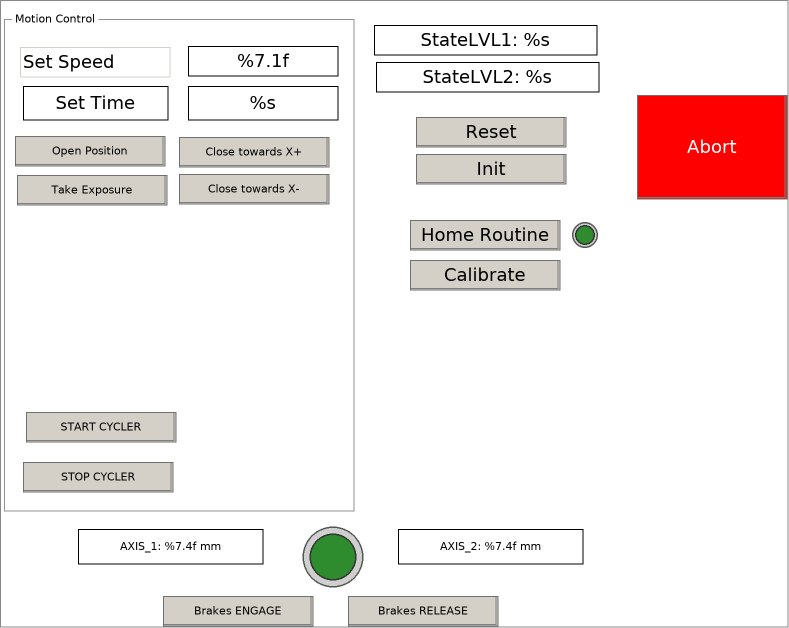
VISUALIZATION ShutterGUI  // 789x628
    GroupBox (4,11 350x500), "Motion Control"
        Rectangle (19,75 145x34), "Set Time", input disabled if: MAIN.shutterFSM.stateLVL2 <> 0;
            OnMouseUp: write GVL.expoTime via Edit, format %7.1f
        Rectangle (184,75 150x34), "%s", text variable: GVL.expoTime
        Button (22,401 150x30), "START CYCLER", input disabled if: MAIN.motionState <> 100;
            OnMouseUp: execute { MAIN.motionState:=3100; }
        Button (19,451 150x30), "STOP CYCLER"
            OnMouseUp: execute { MAIN.stop:=TRUE; }
        Button (13,164 150x30), "Take Exposure", input disabled if: MAIN.shutterFSM.stateLVL2 <> 0;
            OnMouseUp: execute { MAIN.command := commands.takeExposure; }
        Button (11,125 150x30), "Open Position", input disabled if: MAIN.shutterFSM.stateLVL2 <> 0;
            OnMouseUp: execute { MAIN.command := commands.openShutter; }
        Button (175,126 150x30), "Close towards X+", input disabled if: MAIN.shutterFSM.stateLVL2 <> 0;
            OnMouseUp: execute { MAIN.command := commands.closeShutterPX; }
        Button (175,163 150x30), "Close towards X-", input disabled if: MAIN.shutterFSM.stateLVL2 <> 0;
            OnMouseUp: execute { MAIN.command := commands.closeShutterMX; }
    Button (163,596 150x30), "Brakes ENGAGE", input disabled if: MAIN.axis[0].brake=FALSE AND MAIN.axis[1].brake=FALSE;
        OnMouseClick: execute { MAIN.axis[0].brake:=FALSE; MAIN.axis[1].brake:=FALSE; }
    Button (348,596 150x30), "Brakes RELEASE", input disabled if: MAIN.axis[0].brake=TRUE AND MAIN.axis[1].brake=TRUE;
        OnMouseClick: execute { MAIN.axis[0].brake:=TRUE; MAIN.axis[1].brake:=TRUE; }
    Lamp1 (298,522 70x70), variable: MAIN.axis[0].brake and MAIN.axis[1].brake;, style: Lamp-Lamp1-Green
    Rectangle (78,529 185x35), "AXIS_1: %7.4f mm", text variable: MAIN.axis[0].axisRef.NcToPlc.ActPos
    Rectangle (398,529 185x35), "AXIS_2: %7.4f mm", text variable: MAIN.axis[1].axisRef.NcToPlc.ActPos
    Button (416,117 150x30), "Reset"
        OnMouseUp: execute { MAIN.command := commands.clearAllFaults; }
    Button (637,95 150x104), "Abort"
        OnMouseUp: execute { MAIN.command := commands.stopAllMotion; }
    Rectangle (374,25 223x30), "StateLVL1: %s", text variable: MAIN.shutterFSM.stateLVL1;
    Button (410,220 150x30), "Home Routine", input disabled if: MAIN.motionState <> 100;
        OnMouseUp: execute { MAIN.motionState := 400; }
    Textfield (20,47 150x30), "Set Speed", input disabled if: MAIN.shutterFSM.stateLVL2 <> 0;
        OnMouseUp: write MAIN.speed via Default, min 0, max 2000, format %7.1f
    Rectangle (188,46 150x30), "%7.1f", text variable: MAIN.speed
    Lamp1 (570,220 30x30), variable: MAIN.axis[0].axisRef.Status.Homed and MAIN.axis[1].axisRef.Status.Homed;, style: Lamp-Lamp1-Green
    Button (410,260 150x30), "Calibrate", input disabled if: MAIN.motionState <> 100;
        OnMouseUp: execute { MAIN.motionState:=8000; }
    Rectangle (376,62 223x30), "StateLVL2: %s", text variable: MAIN.shutterFSM.stateLVL2;
    Button (416,154 150x30), "Init"
        OnMouseUp: execute { MAIN.command := commands.reinit; }
END_VISUALIZATION

(* stored: Version 1.1.0.1, ProductVersion 3.1.4020.12
   Visu ShutterGUI: Id {1756f6d3-b5ed-4e4e-a9d1-7cd8283dea9e} *)
